// TIA Portal V20 export
// export: Created 2025-12-01T14:57:29.4638747Z, ExportSetting None, DisplayName Totally Integrated Automation Portal, DisplayVersion V20 Update 3, DisplayName TIA Portal Openness, DisplayVersion V20 Update 3, DisplayName TIA Portal Version Control Interface, DisplayVersion V20 Update 3, DisplayName STEP 7 Professional, DisplayVersion V20 Update 3, DisplayName STEP 7 Safety, DisplayVersion V20 Update 2, DisplayName WinCC Basic/Comfort/Advanced, DisplayVersion V20 Update 3, DisplayName WinCC Professional, DisplayVersion V20 Update 3, DisplayName WinCC Unified, DisplayVersion V20 Update 3
FUNCTION "FC78_Errores_CB07" : Void   // FC78, LAD
{ S7_Optimized_Access := 'TRUE' }
// stored: AutoNumber false, SetENOAutomatically false
BEGIN

REGION Network 1: Activacion de los Emergencias
   // 0 seta 1001
   // 1 seta 1010
   // 2 seta 1020
   // 3 seta 1025
   // 4 seta 1029
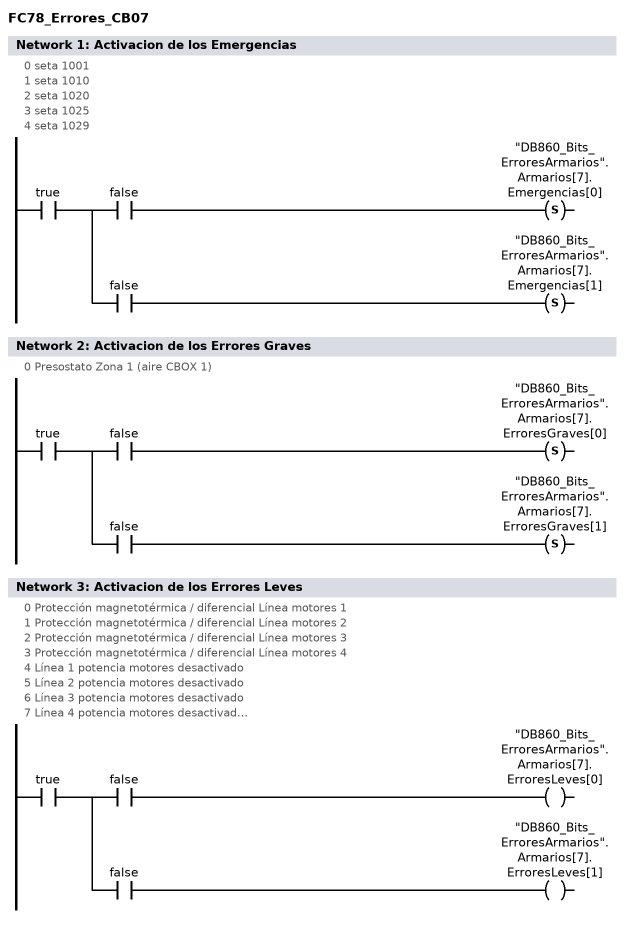
   RUNG wire#powerrail
      Contact( true )
      wire#w1
      Contact( false )
      S_Coil( "DB860_Bits_ErroresArmarios".Armarios[7].Emergencias[0] )
   END_RUNG
   RUNG wire#w1
      Contact( false )
      S_Coil( "DB860_Bits_ErroresArmarios".Armarios[7].Emergencias[1] )
   END_RUNG
   // the same network as SCL:
   IF true AND false THEN
       "DB860_Bits_ErroresArmarios".Armarios[7].Emergencias[0] := TRUE;
       "DB860_Bits_ErroresArmarios".Armarios[7].Emergencias[1] := TRUE;
   END_IF;
END_REGION

REGION Network 2: Activacion de los Errores Graves
   // 0 Presostato Zona 1 (aire CBOX 1)
   RUNG wire#powerrail
      Contact( true )
      wire#w1
      Contact( false )
      S_Coil( "DB860_Bits_ErroresArmarios".Armarios[7].ErroresGraves[0] )
   END_RUNG
   RUNG wire#w1
      Contact( false )
      S_Coil( "DB860_Bits_ErroresArmarios".Armarios[7].ErroresGraves[1] )
   END_RUNG
   // the same network as SCL:
   IF true AND false THEN
       "DB860_Bits_ErroresArmarios".Armarios[7].ErroresGraves[0] := TRUE;
       "DB860_Bits_ErroresArmarios".Armarios[7].ErroresGraves[1] := TRUE;
   END_IF;
END_REGION

REGION Network 3: Activacion de los Errores Leves
   // 0 Protección magnetotérmica / diferencial Línea motores 1
   // 1 Protección magnetotérmica / diferencial Línea motores 2
   // 2 Protección magnetotérmica / diferencial Línea motores 3
   // 3 Protección magnetotérmica / diferencial Línea motores 4
   // 4 Línea 1 potencia motores desactivado
   // 5 Línea 2 potencia motores desactivado
   // 6 Línea 3 potencia motores desactivado
   // 7 Línea 4 potencia motores desactivado
   // 8 Error de nodo profinet barrera medición BarMed_GAL1006 (Nodo 80)
   RUNG wire#powerrail
      Contact( true )
      wire#w1
      Contact( false )
      Coil( "DB860_Bits_ErroresArmarios".Armarios[7].ErroresLeves[0] )
   END_RUNG
   RUNG wire#w1
      Contact( false )
      Coil( "DB860_Bits_ErroresArmarios".Armarios[7].ErroresLeves[1] )
   END_RUNG
   // the same network as SCL:
   "DB860_Bits_ErroresArmarios".Armarios[7].ErroresLeves[0] := true AND false;
   "DB860_Bits_ErroresArmarios".Armarios[7].ErroresLeves[1] := true AND false;
END_REGION
END_FUNCTION
